{attribute 'linkalways'}
{attribute 'hide_all_locals'}
FUNCTION_BLOCK ValueUlint EXTENDS ValueUlintRead IMPLEMENTS Value
VAR
END_VAR

METHOD SetFromType : BOOL
VAR_INPUT
	source : __SYSTEM.AnyType;
END_VAR
SetFromType := ConvertAnyType(source, thisAnyType);
END_METHOD

METHOD SetFromString : BOOL
VAR_INPUT
	value : T_MaxString;
END_VAR
thisValue := STRING_TO_ULINT(value);

SetFromString := TRUE;
END_METHOD

METHOD Set : BOOL
VAR_INPUT
	source : ANY;
END_VAR
Set := ConvertAnyType(source, thisAnyType);
END_METHOD

END_FUNCTION_BLOCK

(* stored: Version 1.1.0.1
   POU ValueUlint: Id {dd582951-0607-4d32-87e2-cce3f481d47b}, SpecialFunc None
   Method SetFromType: Id {15e34f04-9d32-4874-9cbd-689c6875eb8d}
   Method SetFromString: Id {a66b8440-e431-49a3-9951-52e333c55b26}
   Method Set: Id {8d51649c-9006-4e38-91b6-00d687146b61} *)
